// TIA Portal V20 export
// export: Created 2026-07-20T10:18:48.9739534Z, ExportSetting WithDefaults, DisplayName Totally Integrated Automation Portal, DisplayVersion V20 Update 5, DisplayName TIA Portal Openness, DisplayVersion V20 Update 4, DisplayName TIA Portal Version Control Interface, DisplayVersion V20 Update 5, DisplayName SINAMICS Startdrive Advanced, DisplayVersion V20, DisplayName SINAMICS DCC, DisplayVersion V20, DisplayName SINAMICS Startdrive G130, G150, S120, S150, SINAMICS MV, G220, S200, S210, DisplayVersion V20, DisplayName SINAMICS Startdrive G110M, G120, G120C, G120D, G120P, G115D, DisplayVersion V20, DisplayName STEP 7 Professional, DisplayVersion V20 Update 5, DisplayName STEP 7 Safety, DisplayVersion V20 Update 2, DisplayName WinCC Basic/Comfort/Advanced, DisplayVersion V20 Update 5, DisplayName WinCC Unified, DisplayVersion V20 Update 5
FUNCTION "FC_AlarmsMain" : Void   // FC4, LAD
TITLE = Alarms Main
{ S7_Optimized_Access := 'TRUE' }
VERSION : 0.1
// stored: AutoNumber true, IsIECCheckEnabled false, SetENOAutomatically false, UDAEnableTagReadback false
BEGIN

REGION Network 1: Shredder Motor - Fault/Overload Tripped - Check Soft Starter
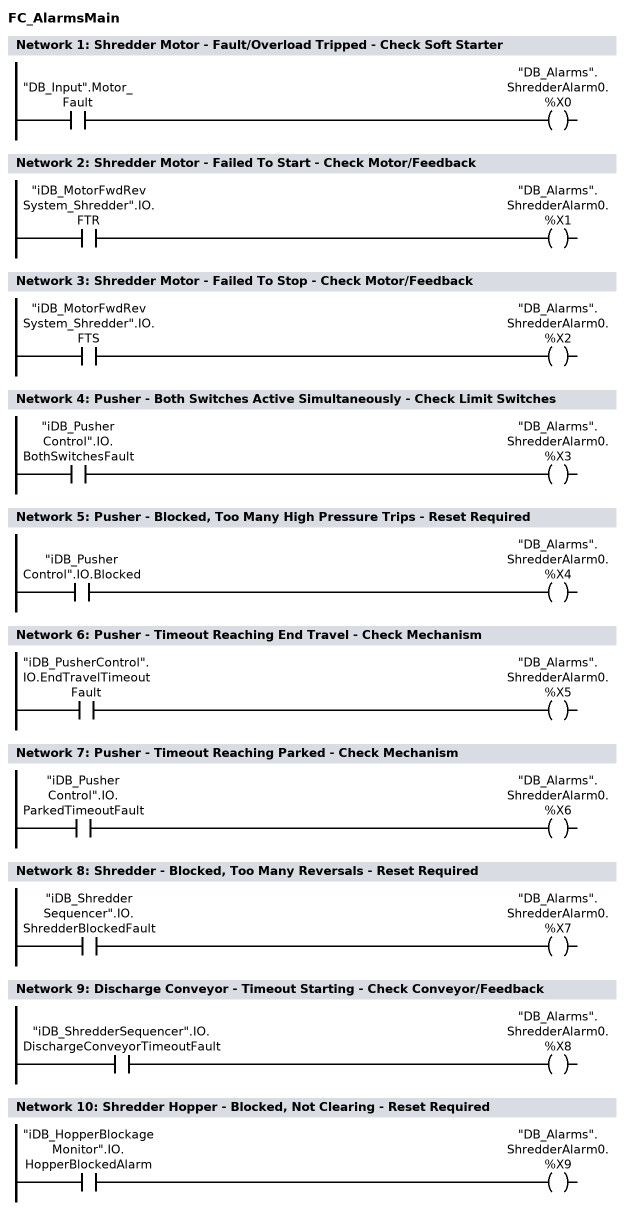
   RUNG wire#powerrail
      Contact( "DB_Input".Motor_Fault )
      Coil( "DB_Alarms".ShredderAlarm0.%X0 )
   END_RUNG
   // the same network as SCL:
   "DB_Alarms".ShredderAlarm0.%X0 := "DB_Input".Motor_Fault;
END_REGION

REGION Network 2: Shredder Motor - Failed To Start - Check Motor/Feedback
   RUNG wire#powerrail
      Contact( "iDB_MotorFwdRevSystem_Shredder".IO.FTR )
      Coil( "DB_Alarms".ShredderAlarm0.%X1 )
   END_RUNG
   // the same network as SCL:
   "DB_Alarms".ShredderAlarm0.%X1 := "iDB_MotorFwdRevSystem_Shredder".IO.FTR;
END_REGION

REGION Network 3: Shredder Motor - Failed To Stop - Check Motor/Feedback
   RUNG wire#powerrail
      Contact( "iDB_MotorFwdRevSystem_Shredder".IO.FTS )
      Coil( "DB_Alarms".ShredderAlarm0.%X2 )
   END_RUNG
   // the same network as SCL:
   "DB_Alarms".ShredderAlarm0.%X2 := "iDB_MotorFwdRevSystem_Shredder".IO.FTS;
END_REGION

REGION Network 4: Pusher - Both Switches Active Simultaneously - Check Limit Switches
   RUNG wire#powerrail
      Contact( "iDB_PusherControl".IO.BothSwitchesFault )
      Coil( "DB_Alarms".ShredderAlarm0.%X3 )
   END_RUNG
   // the same network as SCL:
   "DB_Alarms".ShredderAlarm0.%X3 := "iDB_PusherControl".IO.BothSwitchesFault;
END_REGION

REGION Network 5: Pusher - Blocked, Too Many High Pressure Trips - Reset Required
   RUNG wire#powerrail
      Contact( "iDB_PusherControl".IO.Blocked )
      Coil( "DB_Alarms".ShredderAlarm0.%X4 )
   END_RUNG
   // the same network as SCL:
   "DB_Alarms".ShredderAlarm0.%X4 := "iDB_PusherControl".IO.Blocked;
END_REGION

REGION Network 6: Pusher - Timeout Reaching End Travel - Check Mechanism
   RUNG wire#powerrail
      Contact( "iDB_PusherControl".IO.EndTravelTimeoutFault )
      Coil( "DB_Alarms".ShredderAlarm0.%X5 )
   END_RUNG
   // the same network as SCL:
   "DB_Alarms".ShredderAlarm0.%X5 := "iDB_PusherControl".IO.EndTravelTimeoutFault;
END_REGION

REGION Network 7: Pusher - Timeout Reaching Parked - Check Mechanism
   RUNG wire#powerrail
      Contact( "iDB_PusherControl".IO.ParkedTimeoutFault )
      Coil( "DB_Alarms".ShredderAlarm0.%X6 )
   END_RUNG
   // the same network as SCL:
   "DB_Alarms".ShredderAlarm0.%X6 := "iDB_PusherControl".IO.ParkedTimeoutFault;
END_REGION

REGION Network 8: Shredder - Blocked, Too Many Reversals - Reset Required
   RUNG wire#powerrail
      Contact( "iDB_ShredderSequencer".IO.ShredderBlockedFault )
      Coil( "DB_Alarms".ShredderAlarm0.%X7 )
   END_RUNG
   // the same network as SCL:
   "DB_Alarms".ShredderAlarm0.%X7 := "iDB_ShredderSequencer".IO.ShredderBlockedFault;
END_REGION

REGION Network 9: Discharge Conveyor - Timeout Starting - Check Conveyor/Feedback
   RUNG wire#powerrail
      Contact( "iDB_ShredderSequencer".IO.DischargeConveyorTimeoutFault )
      Coil( "DB_Alarms".ShredderAlarm0.%X8 )
   END_RUNG
   // the same network as SCL:
   "DB_Alarms".ShredderAlarm0.%X8 := "iDB_ShredderSequencer".IO.DischargeConveyorTimeoutFault;
END_REGION

REGION Network 10: Shredder Hopper - Blocked, Not Clearing - Reset Required
   RUNG wire#powerrail
      Contact( "iDB_HopperBlockageMonitor".IO.HopperBlockedAlarm )
      Coil( "DB_Alarms".ShredderAlarm0.%X9 )
   END_RUNG
   // the same network as SCL:
   "DB_Alarms".ShredderAlarm0.%X9 := "iDB_HopperBlockageMonitor".IO.HopperBlockedAlarm;
END_REGION
END_FUNCTION
